TYPE (* a Struct holding 1 Object ID *)
  (* Version 1.0, 2026-05-28, Franz Höpfinger, Demmler Andreas Fahrzeugbau *)
  PACKAGE isobus::UT::Q::types;
  IMPORT isobus::UT::Q::const::IDs::ID_NULL;
  s1ObjectID : STRUCT
    u16ObjId : UINT := ID_NULL; (* Object ID Softkey *)
  END_STRUCT;
END_TYPE
